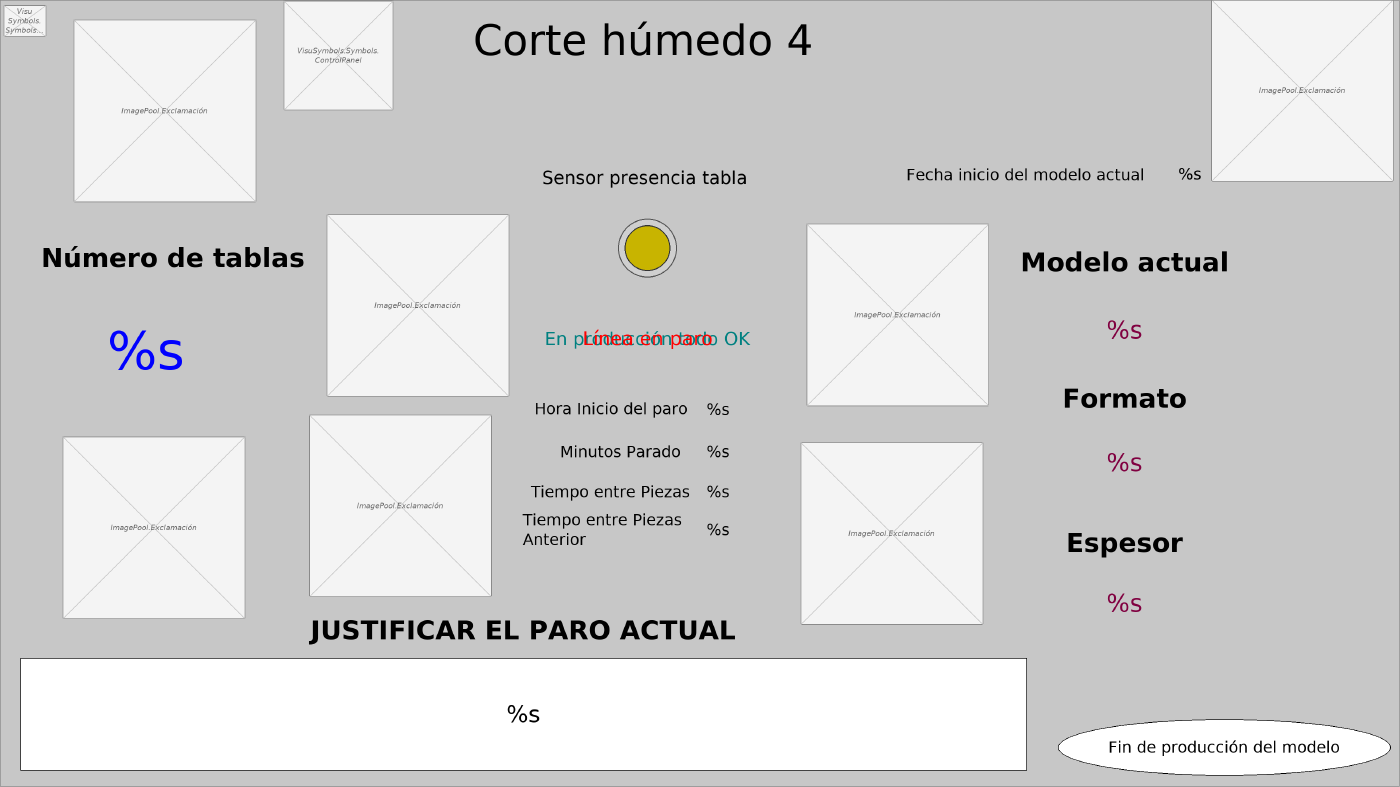
VISUALIZATION Home_CortH4  // 1920x1080
    Ellipse (1451,987 456x77), "Fin de producción del modelo"
        OnMouseClick: OpenDialog Dialog=V_Emerg_Fin_Prod_Ch4, OpenModal=True, OpenCentered=True
    Label (502,0 760x110), "Corte húmedo 4"
    Lamp1 (841,292 94x97), variable: FuncParoNodoCorteH4Remote1.Funci_CortHum4.Fotocelula, style: Lamp-Lamp1-Yellow
    Rectangle (966,547 183x30), "%s", text variable: FuncParoNodoCorteH4Remote1.Funci_CortHum4.H_InParo_Ftc, invisible if: FuncParoNodoCorteH4Remote1.Funci_CortHum4.M_SinParo_Ftc
    Label (730,546 239x30), "Hora Inicio del paro", invisible if: FuncParoNodoCorteH4Remote1.Funci_CortHum4.M_SinParo_Ftc
    Rectangle (966,605 192x30), "%s", text variable: FuncParoNodoCorteH4Remote1.Funci_CortHum4.Min_Parado_Ftc, invisible if: FuncParoNodoCorteH4Remote1.Funci_CortHum4.M_SinParo_Ftc
    Label (765,605 204x30), "Minutos Parado", invisible if: FuncParoNodoCorteH4Remote1.Funci_CortHum4.M_SinParo_Ftc
    Label (725,660 244x30), "Tiempo entre Piezas"
    Label (714,696 255x62), "Tiempo entre Piezas Anterior"
    Rectangle (144,420 183x123), "%s", text variable: FuncParoNodoCorteH4Remote1.Funci_CortHum4.Cont_Piezas_Ftc
    Rectangle (966,660 192x30), "%s", text variable: FuncParoNodoCorteH4Remote1.Funci_CortHum4.t_Entre_Piez_Ftc
    Rectangle (966,712 192x30), "%s", text variable: FuncParoNodoCorteH4Remote1.Funci_CortHum4.t_Entr_Piez_Ante_Ftc
    Label (690,229 397x30), "Sensor presencia tabla"
    Label (725,450 326x30), "En producción todo OK", invisible if: FuncParoNodoCorteH4Remote1.Funci_CortHum4.MParo_Ftc
    Label (771,435 235x59), "Línea en paro", invisible if: FuncParoNodoCorteH4Remote1.Funci_CortHum4.M_SinParo_Ftc
    Label (57,282 361x144), "Número de tablas"
    Label (1362,332 361x56), "Modelo actual"
    Rectangle (1207,426 671x53), "%s", text variable: FuncParoNodoCorteH4Remote1.sModeloActualTabla
    Label (1362,717 361x56), "Espesor"
    Rectangle (1207,801 671x53), "%s", text variable: FuncParoNodoCorteH4Remote1.sEspesorActualTabla
    Label (1362,519 361x56), "Formato"
    Rectangle (1207,608 671x53), "%s", text variable: FuncParoNodoCorteH4Remote1.sFormatoActualTabla
    Rectangle (1613,224 300x30), "%s", text variable: FuncParoNodoCorteH4Remote1.sFechaInicModeloTab
    Label (1240,225 354x30), "Fecha inicio del modelo actual"
    Rectangle (28,903 1380x154), "%s", text variable: FuncParoNodoCorteH4Remote1.Funci_CortHum4.S_Justi_Paro_Ftc, invisible if: FuncParoNodoCorteH4Remote1.Funci_CortHum4.M_SinParo_Ftc
        OnMouseDown: write the text variable via Edit
    Label (27,812 1381x106), "JUSTIFICAR EL PARO ACTUAL", invisible if: FuncParoNodoCorteH4Remote1.Funci_CortHum4.M_SinParo_Ftc
    Image (86,599 250x250), invisible if: FuncParoNodoCorteH4Remote1.Funci_CortHum4.M_SinParo_Ftc, image: ImagePool.Exclamación
    Image (424,569 250x250), invisible if: FuncParoNodoCorteH4Remote1.Funci_CortHum4.M_SinParo_Ftc, image: ImagePool.Exclamación
    Image (1098,607 250x250), invisible if: FuncParoNodoCorteH4Remote1.Funci_CortHum4.M_SinParo_Ftc, image: ImagePool.Exclamación
    Image (101,27 250x250), invisible if: FuncParoNodoCorteH4Remote1.Funci_CortHum4.M_SinParo_Ftc, image: ImagePool.Exclamación
    Image (1106,307 250x250), invisible if: FuncParoNodoCorteH4Remote1.Funci_CortHum4.M_SinParo_Ftc, image: ImagePool.Exclamación
    Image (448,294 250x250), invisible if: FuncParoNodoCorteH4Remote1.Funci_CortHum4.M_SinParo_Ftc, image: ImagePool.Exclamación
    Image (1661,-1 250x250), invisible if: FuncParoNodoCorteH4Remote1.Funci_CortHum4.M_SinParo_Ftc, image: ImagePool.Exclamación
    Image (389,1 150x150), image: VisuSymbols.Symbols.ControlPanel
        OnMouseClick: change screen: Ajustes_CorteH4
    Image (5,7 58x43), image: VisuSymbols.Symbols.Home
        OnMouseClick: change screen: Home_Sel_Maq
END_VISUALIZATION

(* stored: Version 1.1.0.1, ProductVersion 3.1.4024.12
   Visu Home_CortH4: Id {f7a066aa-51fa-41a5-a125-f7a911912ae5} *)
